// TIA Portal V20 export
TYPE "typeCvCoverStatus"
// stored: Access Published, IsFailsafeCompliant true, Namespace Safety
   STRUCT
      cvCoverOK1 { ExternalWritable := 'False'} : Bool;
      cvCoverOK2 { ExternalWritable := 'False'} : Bool;
      cvCoverAllOK { ExternalWritable := 'False'} : Bool;
      cvCoverSystemFaults { ExternalWritable := 'False'} : Bool;
   END_STRUCT;
END_TYPE
